VAR
	stValue: INT;
END_VAR
aRecipeParamsValues[0  ]:= DINT_TO_STRING(stActRecipe.stUBL.nRecipeIndexShow.diValue																		);
aRecipeParamsValues[1  ]:= DINT_TO_STRING(stActRecipe.stUBL.iPackageCapTypeShow.diValue																	);
aRecipeParamsValues[2  ]:= DINT_TO_STRING(stActRecipe.stUBL.iPackageCapDiameterShow.diValue 																);
aRecipeParamsValues[3  ]:= BOOL_TO_STRING(stActRecipe.stUBL.bExEnableShow.bValue 																			);
aRecipeParamsValues[4  ]:= BOOL_TO_STRING(stActRecipe.stUBL.bBottleFeederEnableShow.bValue																);
aRecipeParamsValues[5  ]:= UDINT_TO_STRING(stActRecipe.stUBL.iBottleFeederTurntableVelocitySVShow.udiValue														);
aRecipeParamsValues[6  ]:= DINT_TO_STRING(stActRecipe.stUBL.iBottleFeederBottleSensorDelayShow.diValue													);
aRecipeParamsValues[7  ]:= DINT_TO_STRING(stActRecipe.stUBL.iBottleFeederFormGateDelayShow.diValue														);
aRecipeParamsValues[8  ]:= DINT_TO_STRING(stActRecipe.stUBL.iBottleFeederAllowFormDelayShow.diValue														);
aRecipeParamsValues[9  ]:= BOOL_TO_STRING(stActRecipe.stUBL.bPucksInserterEnableShow.bValue																);
aRecipeParamsValues[10 ]:= UDINT_TO_STRING(stActRecipe.stUBL.iPucksInserterTurntableVelocitySVShow.udiValue 													);
aRecipeParamsValues[11 ]:= UDINT_TO_STRING(stActRecipe.stUBL.iPucksInserterConveyorVelocitySVShow.udiValue														);
aRecipeParamsValues[12 ]:= DINT_TO_STRING(stActRecipe.stUBL.iPucksInserterBottleSensorDelayShow.diValue													);
aRecipeParamsValues[13 ]:= DINT_TO_STRING(stActRecipe.stUBL.iPucksInserterFormGateDelayShow.diValue 														);
aRecipeParamsValues[14 ]:= DINT_TO_STRING(stActRecipe.stUBL.iPucksInserterAllowFormDelayShow.diValue 														);
aRecipeParamsValues[15 ]:= LREAL_TO_STRING(stActRecipe.stUBL.lrPucksInserterWheelOffsetShow.lrValue 															);
aRecipeParamsValues[16 ]:= LREAL_TO_STRING(stActRecipe.stUBL.lrPucksInserterWheelAccelerationShow.lrValue 														);
aRecipeParamsValues[17 ]:= LREAL_TO_STRING(stActRecipe.stUBL.lrPucksInserterWheelVelocityShow.lrValue 															);
aRecipeParamsValues[18 ]:= LREAL_TO_STRING(stActRecipe.stUBL.lrPucksInserterHammerHeightSVShow.lrValue 														);
aRecipeParamsValues[19 ]:= BOOL_TO_STRING(stActRecipe.stUBL.bGateBeforeDispencersEnableShow.bValue														);
aRecipeParamsValues[20 ]:= LREAL_TO_STRING(stActRecipe.stUBL.nGateBeforeDispencersTimeFormInsertingShow.lrValue 												);
aRecipeParamsValues[21 ]:= BOOL_TO_STRING(stActRecipe.stUBL.bGateAfterWeightEnableShow.bValue 															);
aRecipeParamsValues[22 ]:= LREAL_TO_STRING(stActRecipe.stUBL.nGateAfterWeightTimeFormInsertingShow.lrValue 													);
aRecipeParamsValues[25 ]:= BOOL_TO_STRING(stActRecipe.stUBL.bGateRobotEnableShow.bValue       															);
aRecipeParamsValues[26 ]:= LREAL_TO_STRING(stActRecipe.stUBL.nGateRobotTimeFormInsertingShow.lrValue															);
aRecipeParamsValues[27 ]:= BOOL_TO_STRING(stActRecipe.stUBL.bFormsDragingLeftEnableShow.bValue         													);
aRecipeParamsValues[28 ]:= LREAL_TO_STRING(stActRecipe.stUBL.lrFormsDragingLeftVelocityShow.lrValue         													);
aRecipeParamsValues[29 ]:= LREAL_TO_STRING(stActRecipe.stUBL.lrFormsDragingLeftAccelerationShow.lrValue 														);
aRecipeParamsValues[30 ]:= LREAL_TO_STRING(stActRecipe.stUBL.lrFormsDragingLeftDecelerationShow.lrValue   														);
aRecipeParamsValues[31 ]:= BOOL_TO_STRING(stActRecipe.stUBL.bFormsDragingRightEnableShow.bValue 															);
aRecipeParamsValues[32 ]:= LREAL_TO_STRING(stActRecipe.stUBL.lrFormsDragingRightVelocityShow.lrValue 															);
aRecipeParamsValues[33 ]:= LREAL_TO_STRING(stActRecipe.stUBL.lrFormsDragingRightAccelerationShow.lrValue 														);
aRecipeParamsValues[34 ]:= LREAL_TO_STRING(stActRecipe.stUBL.lrFormsDragingRightDecelerationShow.lrValue 														);
aRecipeParamsValues[35 ]:= BOOL_TO_STRING(stActRecipe.stUBL.bDosingTwoPhasesShow.bValue 	        														);
aRecipeParamsValues[36 ]:= LREAL_TO_STRING(stActRecipe.stUBL.lrDispencersLifterReadyPositionShow.lrValue 														);
aRecipeParamsValues[37 ]:= UDINT_TO_STRING(stActRecipe.stUBL.uiDispencerStartDosingDelayShow.udiValue 															);
aRecipeParamsValues[38 ]:= BOOL_TO_STRING(stActRecipe.stUBL.bDispencer1EnableShow.bValue 	          														);
aRecipeParamsValues[39 ]:= BOOL_TO_STRING(stActRecipe.stUBL.bDispencer2EnableShow.bValue 		  															);
aRecipeParamsValues[40 ]:= BOOL_TO_STRING(stActRecipe.stUBL.bDispencer3EnableShow.bValue           														);
aRecipeParamsValues[41 ]:= BOOL_TO_STRING(stActRecipe.stUBL.bDispencer4EnableShow.bValue 			       													);
aRecipeParamsValues[42 ]:= LREAL_TO_STRING(stActRecipe.stUBL.lrDispencer1DoseVolumeShow.lrValue 				   												);
aRecipeParamsValues[43 ]:= LREAL_TO_STRING(stActRecipe.stUBL.lrDispencer1Phase1VolumeShow.lrValue	           													);
aRecipeParamsValues[44 ]:= LREAL_TO_STRING(stActRecipe.stUBL.lrDispencer1Phase2VolumeShow.lrValue 	       														);
aRecipeParamsValues[45 ]:= LREAL_TO_STRING(stActRecipe.stUBL.lrDispencer1Phase1VelocityShow.lrValue 	       													);
aRecipeParamsValues[46 ]:= LREAL_TO_STRING(stActRecipe.stUBL.lrDispencer1Phase2VelocityShow.lrValue 															);
aRecipeParamsValues[47 ]:= LREAL_TO_STRING(stActRecipe.stUBL.lrDispencer1Phase3VelocityShow.lrValue 		   													);
aRecipeParamsValues[48 ]:= LREAL_TO_STRING(stActRecipe.stUBL.lrDispencer1SuckVelocityShow.lrValue   															);
aRecipeParamsValues[49 ]:= LREAL_TO_STRING(stActRecipe.stUBL.lrDispencer1Phase1AccelerationShow.lrValue 														);
aRecipeParamsValues[50 ]:= LREAL_TO_STRING(stActRecipe.stUBL.lrDispencer1Phase2AccelerationShow.lrValue 	  													);
aRecipeParamsValues[51 ]:= LREAL_TO_STRING(stActRecipe.stUBL.lrDispencer1Phase3AccelerationShow.lrValue 	   													);
aRecipeParamsValues[52 ]:= LREAL_TO_STRING(stActRecipe.stUBL.lrDispencer1SuckAccelerationShow.lrValue  														);
aRecipeParamsValues[53 ]:= LREAL_TO_STRING(stActRecipe.stUBL.lrDispencer1Phase1DecelerationShow.lrValue        												);
aRecipeParamsValues[54 ]:= LREAL_TO_STRING(stActRecipe.stUBL.lrDispencer1Phase2DecelerationShow.lrValue 														);
aRecipeParamsValues[55 ]:= LREAL_TO_STRING(stActRecipe.stUBL.lrDispencer1Phase3DecelerationShow.lrValue 	   													);
aRecipeParamsValues[56 ]:= UDINT_TO_STRING(stActRecipe.stUBL.udiDispencer1DosingDoneDelayTimeShow.udiValue 													);
aRecipeParamsValues[57 ]:= LREAL_TO_STRING(stActRecipe.stUBL.lrDispencer1SuckValveOpenVolumeShow.lrValue 														);
aRecipeParamsValues[58 ]:= LREAL_TO_STRING(stActRecipe.stUBL.lrDispencer1SuckValveOpenTimeDelayShow.lrValue 													);
aRecipeParamsValues[59 ]:= LREAL_TO_STRING(stActRecipe.stUBL.lrDispencer1SuckValveCloseVolumeShow.lrValue 														);
aRecipeParamsValues[60 ]:= LREAL_TO_STRING(stActRecipe.stUBL.lrDispencer1SuckValveCloseTimeDelayShow.lrValue 													);
aRecipeParamsValues[61 ]:= LREAL_TO_STRING(stActRecipe.stUBL.lrDispencer1DoseValveOpenVolumeShow.lrValue    													);
aRecipeParamsValues[62 ]:= LREAL_TO_STRING(stActRecipe.stUBL.lrDispencer1DoseValveOpenTimeAccShow.lrValue   													);           						
aRecipeParamsValues[63 ]:= LREAL_TO_STRING(stActRecipe.stUBL.lrDispencer1DoseValveCloseVolumeShow.lrValue    													);           						
aRecipeParamsValues[64 ]:= LREAL_TO_STRING(stActRecipe.stUBL.lrDispencer1DoseValveCloseTimeDecShow.lrValue 													);
aRecipeParamsValues[65 ]:= LREAL_TO_STRING(stActRecipe.stUBL.lrDispencer1DoseSuckingVolumeShow.lrValue 														);
aRecipeParamsValues[66 ]:= LREAL_TO_STRING(stActRecipe.stUBL.lrDispencer1DoseSuckingTimeDelayShow.lrValue 														);
aRecipeParamsValues[67 ]:= BOOL_TO_STRING(stActRecipe.stUBL.bDispencer1DoseSuckingShow.bValue 			       											);
aRecipeParamsValues[68 ]:= BOOL_TO_STRING(stActRecipe.stUBL.bDispencer1LiftSynchroPh1Show.bValue 															);
aRecipeParamsValues[69 ]:= BOOL_TO_STRING(stActRecipe.stUBL.bDispencer1LiftSynchroPh2Show.bValue 			   												);	      							
aRecipeParamsValues[70 ]:= BOOL_TO_STRING(stActRecipe.stUBL.bDispencer1LiftSynchroPh3Show.bValue 		       												);             					
aRecipeParamsValues[71 ]:= LREAL_TO_STRING(stActRecipe.stUBL.lrDispencer1LifterStartDosePositionShow.lrValue													);     						
aRecipeParamsValues[72 ]:= LREAL_TO_STRING(stActRecipe.stUBL.lrDispencer1LifterStopDosePositionShow.lrValue 													);       			
aRecipeParamsValues[73 ]:= LREAL_TO_STRING(stActRecipe.stUBL.lrDispencer1LifterVelocityShow.lrValue            												);	         			
aRecipeParamsValues[74 ]:= LREAL_TO_STRING(stActRecipe.stUBL.lrDispencer1LifterAccelerationShow.lrValue        												);        				
aRecipeParamsValues[75 ]:= LREAL_TO_STRING(stActRecipe.stUBL.lrDispencer1LifterDecelerationShow.lrValue 		    											);              				
aRecipeParamsValues[76 ]:= LREAL_TO_STRING(stActRecipe.stUBL.lrDispencer2DoseVolumeShow.lrValue	            												);              				
aRecipeParamsValues[77 ]:= LREAL_TO_STRING(stActRecipe.stUBL.lrDispencer2Phase1VolumeShow.lrValue 			    												);              				
aRecipeParamsValues[78 ]:= LREAL_TO_STRING(stActRecipe.stUBL.lrDispencer2Phase2VolumeShow.lrValue 			    												);               			
aRecipeParamsValues[79 ]:= LREAL_TO_STRING(stActRecipe.stUBL.lrDispencer2Phase1VelocityShow.lrValue 		    												);               			
aRecipeParamsValues[80 ]:= LREAL_TO_STRING(stActRecipe.stUBL.lrDispencer2Phase2VelocityShow.lrvalue 		    												);               			
aRecipeParamsValues[81 ]:= LREAL_TO_STRING(stActRecipe.stUBL.lrDispencer2Phase3VelocityShow.lrValue 		    												);	      		
aRecipeParamsValues[82 ]:= LREAL_TO_STRING(stActRecipe.stUBL.lrDispencer2SuckVelocityShow.lrValue     															);      				
aRecipeParamsValues[83 ]:= LREAL_TO_STRING(stActRecipe.stUBL.lrDispencer2Phase1AccelerationShow.lrValue 	        											);	         	
aRecipeParamsValues[84 ]:= LREAL_TO_STRING(stActRecipe.stUBL.lrDispencer2Phase2AccelerationShow.lrValue 	        											);         			
aRecipeParamsValues[85 ]:= LREAL_TO_STRING(stActRecipe.stUBL.lrDispencer2Phase3AccelerationShow.lrValue 		    											);	                                        			
aRecipeParamsValues[86 ]:= LREAL_TO_STRING(stActRecipe.stUBL.lrDispencer2SuckAccelerationShow.lrValue   														);                                          			
aRecipeParamsValues[87 ]:= LREAL_TO_STRING(stActRecipe.stUBL.lrDispencer2Phase1DecelerationShow.lrValue 														);                                          			
aRecipeParamsValues[88 ]:= LREAL_TO_STRING(stActRecipe.stUBL.lrDispencer2Phase2DecelerationShow.lrValue 														);            		              			
aRecipeParamsValues[89 ]:= LREAL_TO_STRING(stActRecipe.stUBL.lrDispencer2Phase3DecelerationShow.lrValue 														);           	                			
aRecipeParamsValues[90 ]:= UDINT_TO_STRING(stActRecipe.stUBL.udiDispencer2DosingDoneDelayTimeShow.udiValue 													);                                			
aRecipeParamsValues[91 ]:= LREAL_TO_STRING(stActRecipe.stUBL.lrDispencer2SuckValveOpenVolumeShow.lrValue 														);                               			
aRecipeParamsValues[92 ]:= LREAL_TO_STRING(stActRecipe.stUBL.lrDispencer2SuckValveOpenTimeDelayShow.lrValue 													);                      			
aRecipeParamsValues[93 ]:= LREAL_TO_STRING(stActRecipe.stUBL.lrDispencer2SuckValveCloseVolumeShow.lrValue														);      					
aRecipeParamsValues[94 ]:= LREAL_TO_STRING(stActRecipe.stUBL.lrDispencer2SuckValveCloseTimeDelayShow.lrValue 													);          			
aRecipeParamsValues[95 ]:= LREAL_TO_STRING(stActRecipe.stUBL.lrDispencer2DoseValveOpenVolumeShow.lrValue 														);         			       	
aRecipeParamsValues[96 ]:= LREAL_TO_STRING(stActRecipe.stUBL.lrDispencer2DoseValveOpenTimeAccShow.lrValue 														);					                  	
aRecipeParamsValues[97 ]:= LREAL_TO_STRING(stActRecipe.stUBL.lrDispencer2DoseValveCloseVolumeShow.lrValue 														);					                       	
aRecipeParamsValues[98 ]:= LREAL_TO_STRING(stActRecipe.stUBL.lrDispencer2DoseValveCloseTimeDecShow.lrValue														);					                       	
aRecipeParamsValues[99 ]:= LREAL_TO_STRING(stActRecipe.stUBL.lrDispencer2DoseSuckingVolumeShow.lrValue	    													);					                       	
aRecipeParamsValues[100]:=	LREAL_TO_STRING(stActRecipe.stUBL.lrDispencer2DoseSuckingTimeDelayShow.lrValue														);					                       	
aRecipeParamsValues[101]:=	BOOL_TO_STRING(stActRecipe.stUBL.bDispencer2DoseSuckingShow.bValue 	            											);					                       	
aRecipeParamsValues[102]:=	BOOL_TO_STRING(stActRecipe.stUBL.bDispencer2LiftSynchroPh1Show.bValue 	        												);					
aRecipeParamsValues[103]:=	BOOL_TO_STRING(stActRecipe.stUBL.bDispencer2LiftSynchroPh2Show.bValue 	        												);							
aRecipeParamsValues[104]:=	BOOL_TO_STRING(stActRecipe.stUBL.bDispencer2LiftSynchroPh3Show.bValue 	        												);					    
aRecipeParamsValues[105]:=	LREAL_TO_STRING(stActRecipe.stUBL.lrDispencer2LifterStartDosePositionShow.lrValue													);					    
aRecipeParamsValues[106]:=	LREAL_TO_STRING(stActRecipe.stUBL.lrDispencer2LifterStopDosePositionShow.lrValue 													);					
aRecipeParamsValues[107]:=	LREAL_TO_STRING(stActRecipe.stUBL.lrDispencer2LifterVelocityShow.lrValue        													);					
aRecipeParamsValues[108]:=	LREAL_TO_STRING(stActRecipe.stUBL.lrDispencer2LifterAccelerationShow.lrValue 														);					
aRecipeParamsValues[109]:=	LREAL_TO_STRING(stActRecipe.stUBL.lrDispencer2LifterDecelerationShow.lrValue 	    												);					
aRecipeParamsValues[110]:=	BOOL_TO_STRING(stActRecipe.stUBL.bDispencersCatchEnableShow.bValue             												);					
aRecipeParamsValues[111]:=	BOOL_TO_STRING(stActRecipe.stUBL.bDispencersCatchMaxPressureShow.bValue          												);					
aRecipeParamsValues[112]:=	LREAL_TO_STRING(stActRecipe.stUBL.lrDispencersCatchHeightSVShow.lrValue																);					
aRecipeParamsValues[113]:=	LREAL_TO_STRING(stActRecipe.stUBL.lrDispencersCatch1ClosedValueShow.lrValue          												);					
aRecipeParamsValues[114]:=	LREAL_TO_STRING(stActRecipe.stUBL.lrDispencersCatch1OpenValueShow.lrValue          													);					
aRecipeParamsValues[115]:=	LREAL_TO_STRING(stActRecipe.stUBL.lrDispencersCatch2ClosedValueShow.lrValue       													);						
aRecipeParamsValues[116]:=	LREAL_TO_STRING(stActRecipe.stUBL.lrDispencersCatch2OpenValueShow.lrValue	    													);					 
aRecipeParamsValues[117]:=	LREAL_TO_STRING(stActRecipe.stUBL.lrDispencersCatch3ClosedValueShow.lrValue         												);					
aRecipeParamsValues[118]:=	LREAL_TO_STRING(stActRecipe.stUBL.lrDispencersCatch3OpenValueShow.lrValue           												);					
aRecipeParamsValues[119]:=	LREAL_TO_STRING(stActRecipe.stUBL.lrDispencersCatch4ClosedValueShow.lrValue         												);					
aRecipeParamsValues[120]:=	LREAL_TO_STRING(stActRecipe.stUBL.lrDispencersCatch4OpenValueShow.lrValue															);					
aRecipeParamsValues[121]:=	LREAL_TO_STRING(stActRecipe.stUBL.lrDispencersCatchToleranceShow.lrValue 	        												);					
aRecipeParamsValues[122]:=	BOOL_TO_STRING(stActRecipe.stUBL.bTank1MixerEnableShow.bValue    																); 
aRecipeParamsValues[123]:=	BOOL_TO_STRING(stActRecipe.stUBL.bTankHeatingEnableShow.bValue   																);
aRecipeParamsValues[124]:= DINT_TO_STRING(stActRecipe.stUBL.iTankHeatingTempSVShow.diValue  																);
aRecipeParamsValues[125]:= BOOL_TO_STRING(stActRecipe.stUBL.bTank1PressureEnableShow.bValue																);
aRecipeParamsValues[126]:= BOOL_TO_STRING(stActRecipe.stUBL.bTank1SupplyPumpEnableShow.bValue                             								);
aRecipeParamsValues[127]:= BOOL_TO_STRING(stActRecipe.stUBL.bTank2SupplyPumpEnableShow.bValue                             								);
aRecipeParamsValues[128]:= UDINT_TO_STRING(stActRecipe.stUBL.uTank1LevelSetpointShow.udiValue                              									);
aRecipeParamsValues[129]:= UDINT_TO_STRING(stActRecipe.stUBL.uTank2LevelSetpointShow.udiValue                              									);
aRecipeParamsValues[130]:= BOOL_TO_STRING(stActRecipe.stUBL.bTank1LevelSignalInvertShow.bValue 	                        								);
aRecipeParamsValues[131]:= BOOL_TO_STRING(stActRecipe.stUBL.bTank2LevelSignalInvertShow.bValue 	                        								);
aRecipeParamsValues[132]:= BOOL_TO_STRING(stActRecipe.stUBL.bWeight1EnableShow.bValue                                     								);
aRecipeParamsValues[133]:= LREAL_TO_STRING(stActRecipe.stUBL.lrWeightMassSVShow.lrValue	                                									);
aRecipeParamsValues[134]:= DINT_TO_STRING(stActRecipe.stUBL.iWeight1ActuatorUpDelayShow.diValue 															);
aRecipeParamsValues[135]:= DINT_TO_STRING(stActRecipe.stUBL.iWeight2ActuatorUpDelayShow.diValue                           								);
aRecipeParamsValues[136]:= DINT_TO_STRING(stActRecipe.stUBL.iWeight3ActuatorUpDelayShow.diValue                           								);
aRecipeParamsValues[137]:= DINT_TO_STRING(stActRecipe.stUBL.iWeight4ActuatorUpDelayShow.diValue                           								);
aRecipeParamsValues[138]:= DINT_TO_STRING(stActRecipe.stUBL.iWeight5ActuatorUpDelayShow.diValue                           								);
aRecipeParamsValues[139]:= DINT_TO_STRING(stActRecipe.stUBL.iWeight6ActuatorUpDelayShow.diValue                           								);
aRecipeParamsValues[140]:= LREAL_TO_STRING(stActRecipe.stUBL.lrFormWeightShow.lrValue                                      									);
aRecipeParamsValues[141]:= LREAL_TO_STRING(stActRecipe.stUBL.lrMass1DensityShow.lrValue                                    									);
aRecipeParamsValues[142]:= LREAL_TO_STRING(stActRecipe.stUBL.lrMass2DensityShow.lrValue                                    									);
aRecipeParamsValues[143]:= LREAL_TO_STRING(stActRecipe.stUBL.lrCupWeightShow.lrValue                                       									);
aRecipeParamsValues[144]:= LREAL_TO_STRING(stActRecipe.stUBL.lrWholePackageWeightShow.lrValue 	                            									);
aRecipeParamsValues[145]:= LREAL_TO_STRING(stActRecipe.stUBL.lrWeight1MeasurmentCorrectionShow.lrValue	                    									);
aRecipeParamsValues[146]:= BOOL_TO_STRING(stActRecipe.stUBL.bDispencer1WeightCorrectionEnableShow.bValue                  								);
aRecipeParamsValues[147]:= BOOL_TO_STRING(stActRecipe.stUBL.bDispencer2WeightCorrectionEnableShow.bValue                  								);
aRecipeParamsValues[148]:= BOOL_TO_STRING(stActRecipe.stUBL.bDispencer3WeightCorrectionEnableShow.bValue                  								);
aRecipeParamsValues[149]:= BOOL_TO_STRING(stActRecipe.stUBL.bDispencer4WeightCorrectionEnableShow.bValue                  								);
aRecipeParamsValues[150]:= LREAL_TO_STRING(stActRecipe.stUBL.lrWeightUpperToleranceShow.lrValue                            									);
aRecipeParamsValues[151]:= LREAL_TO_STRING(stActRecipe.stUBL.lrWeightLowerToleranceShow.lrValue                            									);
aRecipeParamsValues[152]:= UDINT_TO_STRING(stActRecipe.stUBL.iWeightCorrectionNumberOfSamplesShow.udiValue                 									);
aRecipeParamsValues[153]:= BOOL_TO_STRING(stActRecipe.stUBL.bLidFeederEnableShow.bValue                 													);
aRecipeParamsValues[154]:= BOOL_TO_STRING(stActRecipe.stUBL.bLidFeederHeaterEnableShow.bValue                             								);
aRecipeParamsValues[155]:= LREAL_TO_STRING(stActRecipe.stUBL.lrLidFeederHeightPosSVShow.lrValue                            									);
aRecipeParamsValues[156]:= DINT_TO_STRING(stActRecipe.stUBL.iLidFeederHeatingTimeShow.diValue                             								);
aRecipeParamsValues[157]:= DINT_TO_STRING(stActRecipe.stUBL.iLidFeederTempHisteresisShow.diValue                          								);
aRecipeParamsValues[158]:= DINT_TO_STRING(stActRecipe.stUBL.iLidFeeder1TempSVShow.diValue 	                            								);
aRecipeParamsValues[159]:= DINT_TO_STRING(stActRecipe.stUBL.iLidFeeder2TempSVShow.diValue 	                            								);
aRecipeParamsValues[160]:= BOOL_TO_STRING(stActRecipe.stUBL.bLidFeederDragingStationEnableShow.bValue 	                								);
aRecipeParamsValues[161]:= LREAL_TO_STRING(stActRecipe.stUBL.lrLidFeederDragingStationVelocityShow.lrValue	                									);
aRecipeParamsValues[162]:= LREAL_TO_STRING(stActRecipe.stUBL.lrLidFeederDragingStationAccelerationShow.lrValue	            									);
aRecipeParamsValues[163]:= LREAL_TO_STRING(stActRecipe.stUBL.lrLidFeederDragingStationDecelerationShow.lrValue	            									);
aRecipeParamsValues[164]:= BOOL_TO_STRING(stActRecipe.stUBL.bLidPuttedCheckEnableShow.bValue                              								);
aRecipeParamsValues[165]:= LREAL_TO_STRING(stActRecipe.stUBL.lrLidPuttedCheckHeightSVShow.lrValue                          									);
aRecipeParamsValues[166]:= LREAL_TO_STRING(stActRecipe.stUBL.lrLidPuttedCheckPositionShow.lrValue                          									);
aRecipeParamsValues[167]:= LREAL_TO_STRING(stActRecipe.stUBL.lrLidPuttedCheckAreaShow.lrValue                              									);
aRecipeParamsValues[168]:= DINT_TO_STRING(stActRecipe.stUBL.iLidPuttedCheckProgramShow.diValue                            								);
aRecipeParamsValues[169]:= BOOL_TO_STRING(stActRecipe.stUBL.bLidSealerEnableShow.bValue                                   								);
aRecipeParamsValues[170]:= BOOL_TO_STRING(stActRecipe.stUBL.bLidSealerHeaterEnableShow.bValue 	                        								);
aRecipeParamsValues[171]:= DINT_TO_STRING(stActRecipe.stUBL.iLidSealerHeatingTimeShow.diValue	                            								);
aRecipeParamsValues[172]:= LREAL_TO_STRING(stActRecipe.stUBL.lrLidSealerPressureShow.lrValue                               									);
aRecipeParamsValues[173]:= LREAL_TO_STRING(stActRecipe.stUBL.lrLidSealerHeightPosSVShow.lrValue                            									);
aRecipeParamsValues[174]:= DINT_TO_STRING(stActRecipe.stUBL.iLidSealerTempHisteresisShow.diValue                          								);
aRecipeParamsValues[175]:= DINT_TO_STRING(stActRecipe.stUBL.iLidSealer1TempSVShow.diValue 	                            								);
aRecipeParamsValues[176]:= DINT_TO_STRING(stActRecipe.stUBL.iLidSealer2TempSVShow.diValue 	                            								);
aRecipeParamsValues[177]:= BOOL_TO_STRING(stActRecipe.stUBL.bLidSealerDragingStationEnableShow.bValue                     								);
aRecipeParamsValues[178]:= LREAL_TO_STRING(stActRecipe.stUBL.lrLidSealerDragingStationVelocityShow.lrValue 	            									);
aRecipeParamsValues[179]:= LREAL_TO_STRING(stActRecipe.stUBL.lrLidSealerDragingStationAccelerationShow.lrValue	            									);
aRecipeParamsValues[180]:= LREAL_TO_STRING(stActRecipe.stUBL.lrLidSealerDragingStationDecelerationShow.lrValue	            									);
aRecipeParamsValues[181]:= BOOL_TO_STRING(stActRecipe.stUBL.bCapFeederGateEnableShow.bValue 	                            								);
aRecipeParamsValues[182]:= DINT_TO_STRING(stActRecipe.stUBL.iCapFeederGateBlockingTimeShow.diValue 	                    								);
aRecipeParamsValues[183]:= BOOL_TO_STRING(stActRecipe.stUBL.bCapFeederEnableShow.bValue                                   								);
aRecipeParamsValues[184]:= LREAL_TO_STRING(stActRecipe.stUBL.lrCapFeederHeightPosSVShow.lrValue                            									);
aRecipeParamsValues[185]:= DINT_TO_STRING(stActRecipe.stUBL.iCapFeederTimeDelayOnShow.diValue                             								);
aRecipeParamsValues[186]:= DINT_TO_STRING(stActRecipe.stUBL.iCapFeederTimeDelayOffShow.diValue                            								);
aRecipeParamsValues[187]:= DINT_TO_STRING(stActRecipe.stUBL.iCapFeederTimeToEmptySleeveErrorShow.diValue                  								);
aRecipeParamsValues[188]:= BOOL_TO_STRING(stActRecipe.stUBL.bCapSorterOnlyWeightOKEnableShow.bValue                       								);
aRecipeParamsValues[189]:= BOOL_TO_STRING(stActRecipe.stUBL.bCapSorterDragEnableShow.bValue                               								);
aRecipeParamsValues[190]:= LREAL_TO_STRING(stActRecipe.stUBL.lrCapSorterDragVelocityShow.lrValue                           									);
aRecipeParamsValues[191]:= LREAL_TO_STRING(stActRecipe.stUBL.lrCapSorterDragAccelerationShow.lrValue 	                    									);
aRecipeParamsValues[192]:= LREAL_TO_STRING(stActRecipe.stUBL.lrCapSorterDragDecelerationShow.lrValue 	                    									);
aRecipeParamsValues[193]:= BOOL_TO_STRING(stActRecipe.stUBL.bCapPuttedCheckEnableShow.bValue                              								);
aRecipeParamsValues[194]:= LREAL_TO_STRING(stActRecipe.stUBL.lrCapPuttedCheckHeightPosSVShow.lrValue 	                    									);
aRecipeParamsValues[195]:= BOOL_TO_STRING(stActRecipe.stUBL.bGripperScrewer1EnableShow.bValue 	                        								);
aRecipeParamsValues[196]:= LREAL_TO_STRING(stActRecipe.stUBL.lrGripperScrewingTightTorqueShow.lrValue                      									);
aRecipeParamsValues[197]:= BOOL_TO_STRING(stActRecipe.stUBL.bGripperScrewer2EnableShow.bValue 	                        								);
aRecipeParamsValues[198]:= LREAL_TO_STRING(stActRecipe.stUBL.lrGripperScrewing2TightTorqueShow.lrValue	                    									);
aRecipeParamsValues[199]:= DINT_TO_STRING(stActRecipe.stUBL.iGripperScrewer1ToolShow.diValue                              								);
aRecipeParamsValues[200]:= LREAL_TO_STRING(stActRecipe.stUBL.lrGripperScrewer1VelocityShow.lrValue                         									);
aRecipeParamsValues[201]:= DINT_TO_STRING(stActRecipe.stUBL.nGripperScrewer1TightTimeShow.diValue	                        								);
aRecipeParamsValues[202]:= DINT_TO_STRING(stActRecipe.stUBL.iGripperScrewer1StartDelayShow.diValue	                    								);
aRecipeParamsValues[203]:= LREAL_TO_STRING(stActRecipe.stUBL.lrGripperScrewerReadyPositionShow.lrValue 	                									);
aRecipeParamsValues[204]:= LREAL_TO_STRING(stActRecipe.stUBL.lrGripperScrewerPushingCapPositionShow.lrValue 	            									);
aRecipeParamsValues[205]:= LREAL_TO_STRING(stActRecipe.stUBL.lrGripperScrewerScrewingCapPositionShow.lrValue               									);
aRecipeParamsValues[206]:= LREAL_TO_STRING(stActRecipe.stUBL.lrGripperScrewerPressureShow.lrValue                          									);
aRecipeParamsValues[207]:= LREAL_TO_STRING(stActRecipe.stUBL.lrGripperScrewerCatchPressureShow.lrValue 	                									);
aRecipeParamsValues[208]:= LREAL_TO_STRING(stActRecipe.stUBL.lrDispencerCatchPressureShow.lrValue                          									);
aRecipeParamsValues[209]:= LREAL_TO_STRING(stActRecipe.stUBL.lrGripperScrewerPressureExhaustLevelShow.lrValue              									);
aRecipeParamsValues[210]:= LREAL_TO_STRING(stActRecipe.stUBL.lrGripperScrewerCatchPressureExhaustLevelShow.lrValue         									);
aRecipeParamsValues[211]:= LREAL_TO_STRING(stActRecipe.stUBL.lrGripperScrewerTurnoversToFullScrewedShow.lrValue 	        									);
aRecipeParamsValues[212]:= LREAL_TO_STRING(stActRecipe.stUBL.lrGripperScrewerThreadPitchShow.lrValue                       									);
aRecipeParamsValues[213]:= LREAL_TO_STRING(stActRecipe.stUBL.lrGripperScrewerThreadTimesShow.lrValue                       									);
aRecipeParamsValues[214]:= DINT_TO_STRING(stActRecipe.stUBL.nGripperScrewerCatchHeightSVShow.diValue	                    								);
aRecipeParamsValues[215]:= BOOL_TO_STRING(stActRecipe.stUBL.bGripperScrewer1FindScrewShow.bValue                          								);
aRecipeParamsValues[216]:= BOOL_TO_STRING(stActRecipe.stUBL.bGripperScrewer1Option4Show.bValue                            								);
aRecipeParamsValues[217]:= LREAL_TO_STRING(stActRecipe.stUBL.lrGripperScrewer1FindingScrewDegreeShow.lrValue               									);
aRecipeParamsValues[218]:= BOOL_TO_STRING(stActRecipe.stUBL.bGripperScrewer1Option1Show.bValue	                        								);
aRecipeParamsValues[219]:= BOOL_TO_STRING(stActRecipe.stUBL.bGripperScrewer1Option2Show.bValue	                        								);
aRecipeParamsValues[220]:= BOOL_TO_STRING(stActRecipe.stUBL.bGripperScrewer1Option3Show.bValue	                        								);
aRecipeParamsValues[221]:= BOOL_TO_STRING(stActRecipe.stUBL.bGripperScrewer1Option5Show.bValue	                        								);
aRecipeParamsValues[222]:= BOOL_TO_STRING(stActRecipe.stUBL.bGripperScrewer1Option6Show.bValue	                        								);
aRecipeParamsValues[223]:= BOOL_TO_STRING(stActRecipe.stUBL.bGripperScrewer1Option7Show.bValue	                        								);
aRecipeParamsValues[224]:= BOOL_TO_STRING(stActRecipe.stUBL.bBottleDragingStationEnableShow.bValue 	                    								);
aRecipeParamsValues[225]:= LREAL_TO_STRING(stActRecipe.stUBL.lrBottleDragingStationVelocityShow.lrValue                    									);
aRecipeParamsValues[226]:= BOOL_TO_STRING(stActRecipe.stUBL.bCapCorrectCheckEnableShow.bValue 	                        								);
aRecipeParamsValues[227]:= LREAL_TO_STRING(stActRecipe.stUBL.lrCapCorrectCheckHeightPosSVShow.lrValue                      									);
aRecipeParamsValues[228]:= BOOL_TO_STRING(stActRecipe.stUBL.bCapCorrectCheckCameraEnableShow.bValue                       								);
aRecipeParamsValues[229]:= DINT_TO_STRING(stActRecipe.stUBL.iCapCorrectCheckCameraProgramShow.diValue 	                								);
aRecipeParamsValues[230]:= BOOL_TO_STRING(stActRecipe.stUBL.bBottleTransferEnableShow.bValue			                    								);
aRecipeParamsValues[231]:= UDINT_TO_STRING(stActRecipe.stUBL.nBottleTransferProgramShow.udiValue			                									);
aRecipeParamsValues[232]:= DINT_TO_STRING(stActRecipe.stUBL.iBottleTransferPickOffsetXShow.diValue                        								);
aRecipeParamsValues[233]:= DINT_TO_STRING(stActRecipe.stUBL.iBottleTransferPickOffsetYShow.diValue 	                    								);
aRecipeParamsValues[234]:= DINT_TO_STRING(stActRecipe.stUBL.iBottleTransferPickOffsetZShow.diValue                        								);
aRecipeParamsValues[235]:= DINT_TO_STRING(stActRecipe.stUBL.iBottleTransferPick2OffsetXShow.diValue                       								);
aRecipeParamsValues[236]:= DINT_TO_STRING(stActRecipe.stUBL.iBottleTransferPick2OffsetYShow.diValue 	                    								);
aRecipeParamsValues[237]:= DINT_TO_STRING(stActRecipe.stUBL.iBottleTransferPick2OffsetZShow.diValue                       								);
aRecipeParamsValues[238]:= DINT_TO_STRING(stActRecipe.stUBL.iBottleTransferPlace1OffsetXShow.diValue 	                    								);
aRecipeParamsValues[239]:= DINT_TO_STRING(stActRecipe.stUBL.iBottleTransferPlace1OffsetYShow.diValue 	                    								);
aRecipeParamsValues[240]:= DINT_TO_STRING(stActRecipe.stUBL.iBottleTransferPlace1OffsetZShow.diValue 	                    								);
aRecipeParamsValues[241]:= DINT_TO_STRING(stActRecipe.stUBL.iBottleTransferPlace2OffsetXShow.diValue 	                    								);
aRecipeParamsValues[242]:= DINT_TO_STRING(stActRecipe.stUBL.iBottleTransferPlace2OffsetYShow.diValue 	                    								);
aRecipeParamsValues[243]:= DINT_TO_STRING(stActRecipe.stUBL.iBottleTransferPlace2OffsetZShow.diValue 	                    								);
aRecipeParamsValues[244]:=	DINT_TO_STRING(stActRecipe.stUBL.iBottleTransferSpeedShow.diValue 	                            								);
aRecipeParamsValues[245]:= BOOL_TO_STRING(stActRecipe.stUBL.bBottleTransferInkJetEnableShow.bValue 	                    								);
aRecipeParamsValues[246]:= BOOL_TO_STRING(stActRecipe.stUBL.bBottleTransferPickOnlyOneShow.bValue                         								);
aRecipeParamsValues[247]:= BOOL_TO_STRING(stActRecipe.stUBL.bBottleTransferWeightEnableShow.bValue 	                    								);
aRecipeParamsValues[248]:= DINT_TO_STRING(stActRecipe.stUBL.iBottleTransferWeightIntervalShow.diValue	                    								);
aRecipeParamsValues[249]:= BOOL_TO_STRING(stActRecipe.stUBL.bBottleTransferRotateEnableShow.bValue 	                    								);
aRecipeParamsValues[250]:= BOOL_TO_STRING(stActRecipe.stUBL.bBadBottleConveyorEnableShow.bValue                           								);
aRecipeParamsValues[251]:= UDINT_TO_STRING(stActRecipe.stUBL.nBadBottleConveyorVelocitySVShow.udiValue 	                									);
aRecipeParamsValues[252]:= BOOL_TO_STRING(stActRecipe.stUBL.bLabelMachineEnableShow.bValue 	                            								);
aRecipeParamsValues[253]:= BOOL_TO_STRING(stActRecipe.stUBL.bExitTurnTable1EnableShow.bValue                              								);
aRecipeParamsValues[254]:= BOOL_TO_STRING(stActRecipe.stUBL.bExitConveyorEnableShow.bValue                                								);
aRecipeParamsValues[255]:= UDINT_TO_STRING(stActRecipe.stUBL.nExitConveyorVelocitySVShow.udiValue 	                        									);
aRecipeParamsValues[256]:= BOOL_TO_STRING(stActRecipe.stUBL.bFormTransportersEnableShow.bValue						    								);
aRecipeParamsValues[257]:= UDINT_TO_STRING(stActRecipe.stUBL.nFormTransportersDispencerVelocitySVShow.udiValue	            									);
aRecipeParamsValues[258]:= UDINT_TO_STRING(stActRecipe.stUBL.nFormTransportersScrewerVelocitySVShow.udiValue			    									);
aRecipeParamsValues[259]:= UDINT_TO_STRING(stActRecipe.stUBL.nFormTransportersBeforeScrewerVelocitySVShow.udiValue	        									);
aRecipeParamsValues[260]:= UDINT_TO_STRING(stActRecipe.stUBL.nFormTransportersSlowerVelocitySVShow.udiValue		 	    									);
aRecipeParamsValues[261]:= BOOL_TO_STRING(stActRecipe.stUBL.bCircularInkjetEnableShow.bValue	 	                        								);
aRecipeParamsValues[262]:= DINT_TO_STRING(stActRecipe.stUBL.iCircularInkjetSpeedShow.diValue	 	                        								);
aRecipeParamsValues[263]:= DINT_TO_STRING(stActRecipe.stUBL.iCircularInkjetDelayShow.diValue	 	                        								);
aRecipeParamsValues[264]:= DINT_TO_STRING(stActRecipe.stUBL.iCircularInkjetHoldShow.diValue	 	                        								);
aRecipeParamsValues[265]:= DINT_TO_STRING(stActRecipe.stUCF.iCapSorterProductType.diValue 	                            								);
aRecipeParamsValues[266]:= UDINT_TO_STRING(stActRecipe.stUCF.uiCapSorterIndexShow.udiValue 																	);
aRecipeParamsValues[267]:= BOOL_TO_STRING(stActRecipe.stUCF.bPresenceBottleEnableShow.bValue 	                            								);
aRecipeParamsValues[268]:= BOOL_TO_STRING(stActRecipe.stUCF.bCapSorterTransporterEnableShow.bValue														);
aRecipeParamsValues[269]:= DINT_TO_STRING(stActRecipe.stUCF.iCapSorterTransporterTankConveyorVelocityShow.diValue											);
aRecipeParamsValues[270]:= DINT_TO_STRING(stActRecipe.stUCF.iCapSorterTransporterStartDelayTimeShow.diValue												);
aRecipeParamsValues[271]:= UDINT_TO_STRING(stActRecipe.stUCF.udiCapSorterTransporterTimeProductOnSensorBeforeBrushShow.udiValue								);
aRecipeParamsValues[272]:= DINT_TO_STRING(stActRecipe.stUCF.iCapSorterTransporterEmptyingConveyorSpeedShow.diValue										);
aRecipeParamsValues[273]:= DINT_TO_STRING(stActRecipe.stUCF.iCapSorterTransporterVolumeOfCapsShow.diValue													);
aRecipeParamsValues[274]:= BOOL_TO_STRING(stActRecipe.stUCF.bCapSorterWheelEnableShow.bValue							    								);
aRecipeParamsValues[275]:= LREAL_TO_STRING(stActRecipe.stUCF.lrCapSorterWheelMoveAccelerationEmptyTableShow.lrValue	    									);
aRecipeParamsValues[276]:= LREAL_TO_STRING(stActRecipe.stUCF.lrCapSorterWheelMoveDecelerationEmptyTableShow.lrValue	    									);
aRecipeParamsValues[277]:= LREAL_TO_STRING(stActRecipe.stUCF.lrCapSorterWheelMoveSpeedEmptyTableShow.lrValue			    									);
aRecipeParamsValues[278]:= LREAL_TO_STRING(stActRecipe.stUCF.lrCapSorterWheelMoveAngleEmptyTableShow.lrValue			    									);
aRecipeParamsValues[279]:= LREAL_TO_STRING(stActRecipe.stUCF.lrCapSorterWheelJerkAngleEmptyTableShow.lrValue			    									);
aRecipeParamsValues[280]:= DINT_TO_STRING(stActRecipe.stUCF.iCapSorterWheelWaitingAfterRotationEmptyTableShow.diValue     								);
aRecipeParamsValues[281]:= LREAL_TO_STRING(stActRecipe.stUCF.lrCapSorterWheelMoveAccelerationFullTableShow.lrValue	        									);
aRecipeParamsValues[282]:= LREAL_TO_STRING(stActRecipe.stUCF.lrCapSorterWheelMoveDecelerationFullTableShow.lrValue	        									);
aRecipeParamsValues[283]:= LREAL_TO_STRING(stActRecipe.stUCF.lrCapSorterWheelMoveSpeedFullTableShow.lrValue			    									);
aRecipeParamsValues[284]:= LREAL_TO_STRING(stActRecipe.stUCF.lrCapSorterWheelMoveAngleFullyTableShow.lrValue			    									);
aRecipeParamsValues[285]:= LREAL_TO_STRING(stActRecipe.stUCF.lrCapSorterWheelJerkAngleFullTableShow.lrValue			    									);
aRecipeParamsValues[286]:= DINT_TO_STRING(stActRecipe.stUCF.iCapSorterWheelWaitingAfterRotationFullTableShow.diValue      								);
aRecipeParamsValues[287]:= LREAL_TO_STRING(stActRecipe.stUCF.lrCapSorterWheelMoveAccelerationHalfFullTableShow.lrValue     									);
aRecipeParamsValues[288]:= LREAL_TO_STRING(stActRecipe.stUCF.lrCapSorterWheelMoveDecelerationHalfFullTableShow.lrValue     									);
aRecipeParamsValues[289]:= LREAL_TO_STRING(stActRecipe.stUCF.lrCapSorterWheelMoveSpeedHalfFullTableShow.lrValue												);
aRecipeParamsValues[290]:= LREAL_TO_STRING(stActRecipe.stUCF.lrCapSorterWheelMoveAngleHalfFullyTableShow.lrValue												);
aRecipeParamsValues[291]:= LREAL_TO_STRING(stActRecipe.stUCF.lrCapSorterWheelJerkAngleHalfFullTableShow.lrValue												);
aRecipeParamsValues[292]:= DINT_TO_STRING(stActRecipe.stUCF.iCapSorterWheelWaitingAfterRotationHalfFullTableShow.diValue 									);
aRecipeParamsValues[293]:= BOOL_TO_STRING(stActRecipe.stUCF.bCapSorterCameraEnableShow.bValue                            									);
aRecipeParamsValues[294]:= BOOL_TO_STRING(stActRecipe.stUCF.bCapSorterRobotEnableShow.bValue                 			    								);
aRecipeParamsValues[295]:= LREAL_TO_STRING(stActRecipe.stUCF.lrCapSorterRobotPlace1PositionXShow.lrValue														);
aRecipeParamsValues[296]:= LREAL_TO_STRING(stActRecipe.stUCF.lrCapSorterRobotPlace1PositionYShow.lrValue														);
aRecipeParamsValues[297]:= LREAL_TO_STRING(stActRecipe.stUCF.lrCapSorterRobotPlace1PositionZShow.lrValue														);
aRecipeParamsValues[298]:= LREAL_TO_STRING(stActRecipe.stUCF.lrCapSorterRobotPlace1PositionCShow.lrValue														);
aRecipeParamsValues[299]:= DINT_TO_STRING(stActRecipe.stUCF.iCapSorterRobotPickElevationShow.diValue														);
aRecipeParamsValues[300]:= DINT_TO_STRING(stActRecipe.stUCF.iCapSorterRobotPickTimeShow.diValue															);
aRecipeParamsValues[301]:= DINT_TO_STRING(stActRecipe.stUCF.iCapSorterRobotVacuumActivationShow.diValue													);
aRecipeParamsValues[302]:= DINT_TO_STRING(stActRecipe.stUCF.iCapSorterRobotVacuumOffShow.diValue						    								);
aRecipeParamsValues[303]:= DINT_TO_STRING(stActRecipe.stUCF.iCapSorterRobotPlaceTimeShow.diValue															);
aRecipeParamsValues[304]:= DINT_TO_STRING(stActRecipe.stUCF.iCapSorterRobotTCP_PlaceOffsetShow.diValue			    									);
aRecipeParamsValues[305]:= DINT_TO_STRING(stActRecipe.stUCF.iCapSorterRobotAccelerationDecelerationShow.diValue	 										);
aRecipeParamsValues[306]:= DINT_TO_STRING(stActRecipe.stUCF.iCapSorterRobotGripperWatchdogShow.diValue			    									);
aRecipeParamsValues[307]:= DINT_TO_STRING(stActRecipe.stUCF.iCapSorterRobotParalaxCorrectionShow.diValue		    										);
aRecipeParamsValues[308]:= DINT_TO_STRING(stActRecipe.stUCF.iCapSorterRobotNumberToolShow.diValue		 													);
aRecipeParamsValues[309]:= DINT_TO_STRING(stActRecipe.stUCF.iCapSorterRobotPickPositionZShow.diValue 														);
aRecipeParamsValues[310]:= DINT_TO_STRING(stActRecipe.stUCF.iCapSorterRobotTCP_Lenght.diValue		 														);
aRecipeParamsValues[311]:= DINT_TO_STRING(stActRecipe.stUCF.iCapSorterRobotProductDiametr.diValue	 														);
aRecipeParamsValues[312]:= BOOL_TO_STRING(stActRecipe.stUCF.bCapSorterIntermediateTransporterEnableShow.bValue											);
aRecipeParamsValues[313]:= DINT_TO_STRING(stActRecipe.stUCF.iCapSorterIntermediateTransporterAutoSpeedShow.diValue										);
aRecipeParamsValues[314]:= DINT_TO_STRING(stActRecipe.stUCF.iCapSorterIntermediateTransporterManualSpeedShow.diValue										);
aRecipeParamsValues[315]:= DINT_TO_STRING(stActRecipe.stUCF.iCapSorterIntermediateTransporterEmptyingSpeedShow.diValue									);
aRecipeParamsValues[316]:= DINT_TO_STRING(stActRecipe.stUCF.iCapSorterIntermediateTransporterDelayCountTimeShow.diValue									);
aRecipeParamsValues[317]:= DINT_TO_STRING(stActRecipe.stUCF.iCapSorterIntermediateTransporterReverseTimeShow.diValue										);
aRecipeParamsValues[318]:= UDINT_TO_STRING(stActRecipe.stUCF.udiCapSorterIntermediateTransporterTimeProductOnSensorShow.udiValue 								);
aRecipeParamsValues[319]:= LREAL_TO_STRING(stActRecipe.stUCF.lrCapSorterIntermediateTransporterWheelAngleShow.lrValue											);
aRecipeParamsValues[320]:= BOOL_TO_STRING(stActRecipe.stUCF.bCapSorterIntermediateBrushEnableShow.bValue			 	    								);
aRecipeParamsValues[321]:= DINT_TO_STRING(stActRecipe.stUCF.iCapSorterIntermediateBrushAutoSpeedShow.diValue		 	    								);
aRecipeParamsValues[322]:= DINT_TO_STRING(stActRecipe.stUCF.iCapSorterIntermediateBrushManualSpeedShow.diValue		  									);
aRecipeParamsValues[323]:= DINT_TO_STRING(stActRecipe.stUCF.iCapSorterIntermediateBrushEmptyingSpeedShow.diValue	 	    								);
aRecipeParamsValues[324]:= LREAL_TO_STRING(stActRecipe.stUCF.lrCapSorterIntermediateBrushPositionHeightSVShow.lrValue 											);
aRecipeParamsValues[325]:= BOOL_TO_STRING(stActRecipe.stUCF.bCapSorterBrush1OnWheelEnableShow.bValue			  											);
aRecipeParamsValues[326]:= DINT_TO_STRING(stActRecipe.stUCF.iCapSorterBrush1OnWheelAutoSpeedShow.diValue		  											);
aRecipeParamsValues[327]:= DINT_TO_STRING(stActRecipe.stUCF.iCapSorterBrush1OnWheelManualSpeedShow.diValue		     									);
aRecipeParamsValues[328]:= DINT_TO_STRING(stActRecipe.stUCF.iCapSorterBrush1OnWheelEmptyingSpeedShow.diValue	  											);
aRecipeParamsValues[329]:= LREAL_TO_STRING(stActRecipe.stUCF.lrCapSorterBrush1OnWheelPositionHeightSVShow.lrValue   											);
aRecipeParamsValues[330]:= BOOL_TO_STRING(stActRecipe.stUCF.bCapSorterBrush2OnWheelEnableShow.bValue			 											);
aRecipeParamsValues[331]:= DINT_TO_STRING(stActRecipe.stUCF.iCapSorterBrush2OnWheelAutoSpeedShow.diValue		 											);
aRecipeParamsValues[332]:= DINT_TO_STRING(stActRecipe.stUCF.iCapSorterBrush2OnWheelManualSpeedShow.diValue	      										);
aRecipeParamsValues[333]:= DINT_TO_STRING(stActRecipe.stUCF.iCapSorterBrush2OnWheelEmptyingSpeedShow.diValue	   											);
aRecipeParamsValues[334]:= LREAL_TO_STRING(stActRecipe.stUCF.lrCapSorterBrush2OnWheelPositionHeightSVShow.lrValue   											);
aRecipeParamsValues[335]:= BOOL_TO_STRING(stActRecipe.stUCF.bCapSorterFeederEnableShow.bValue																);
aRecipeParamsValues[336]:= BOOL_TO_STRING(stActRecipe.stUCF.bCapSorterFeederEnableTubeError.bValue														);
aRecipeParamsValues[337]:= LREAL_TO_STRING(stActRecipe.stUCF.lrCapSorterFeederMover1InputPositionShow.lrValue													);
aRecipeParamsValues[338]:= LREAL_TO_STRING(stActRecipe.stUCF.lrCapSorterFeederMover2InputPositionShow.lrValue													);
aRecipeParamsValues[339]:= LREAL_TO_STRING(stActRecipe.stUCF.lrCapSorterFeederMover1OutputPositionShow.lrValue													);
aRecipeParamsValues[340]:= LREAL_TO_STRING(stActRecipe.stUCF.lrCapSorterFeederMover2OutputPositionShow.lrValue													);
aRecipeParamsValues[341]:= LREAL_TO_STRING(stActRecipe.stUCF.lrCapSorterFeederSlotDistanceShow.lrValue															);
aRecipeParamsValues[342]:= LREAL_TO_STRING(stActRecipe.stUCF.lrCapSorterFeederMoverSpeedShow.lrValue															);
aRecipeParamsValues[343]:= LREAL_TO_STRING(stActRecipe.stUCF.lrCapSorterFeederMoverAccelerationShow.lrValue    												);
aRecipeParamsValues[344]:= LREAL_TO_STRING(stActRecipe.stUCF.lrCapSorterFeederMoveJerkShow.lrValue																);
aRecipeParamsValues[345]:= BOOL_TO_STRING(stActRecipe.stUCF.bCapSorterPreScrewerEnableShow.bValue															);
aRecipeParamsValues[346]:= BOOL_TO_STRING(stActRecipe.stUCF.bCapSorterPreScrewerPicker1EnableShow.bValue           										);
aRecipeParamsValues[347]:= BOOL_TO_STRING(stActRecipe.stUCF.bCapSorterPreScrewerPicker2EnableShow.bValue           										);
aRecipeParamsValues[348]:= BOOL_TO_STRING(stActRecipe.stUCF.bCapSorterPreScrewerPicker3EnableShow.bValue          										);
aRecipeParamsValues[349]:= BOOL_TO_STRING(stActRecipe.stUCF.bCapSorterPreScrewerPicker4EnableShow.bValue          										);
aRecipeParamsValues[350]:= LREAL_TO_STRING(stActRecipe.stUCF.lrCapSorterPreScrewerPickZPositionShow.lrValue													);
aRecipeParamsValues[351]:= LREAL_TO_STRING(stActRecipe.stUCF.lrCapSorterPreScrewerCatcherReleseShow.lrValue													);
aRecipeParamsValues[352]:= LREAL_TO_STRING(stActRecipe.stUCF.lrCapSorterPreScrewerCapCatcherZPositionShow.lrValue												);
aRecipeParamsValues[353]:= LREAL_TO_STRING(stActRecipe.stUCF.lrCapSorterPreScrewerTopZPositionShow.lrValue														);
aRecipeParamsValues[354]:= LREAL_TO_STRING(stActRecipe.stUCF.lrCapSorterPreScrewerCartesianCatchZPositionShow.lrValue											);
aRecipeParamsValues[355]:= LREAL_TO_STRING(stActRecipe.stUCF.lrCapSorterPreScrewerStrawCatcherZPositionShow.lrValue											);
aRecipeParamsValues[356]:= LREAL_TO_STRING(stActRecipe.stUCF.LrCapSorterPreScrewerCheckStrawCatcherActuatorZPosition.lrValue 									);
aRecipeParamsValues[357]:= LREAL_TO_STRING(stActRecipe.stUCF.lrCapSorterPreScrewerScrewerStartZPositionShow.lrValue											);
aRecipeParamsValues[358]:= LREAL_TO_STRING(stActRecipe.stUCF.lrCapSorterPreScrewerGripperOpenPositionShow.lrValue												);
aRecipeParamsValues[359]:= LREAL_TO_STRING(stActRecipe.stUCF.lrCapSorterPreScrewerPlaceZPositionShow.lrValue													);
aRecipeParamsValues[360]:= LREAL_TO_STRING(stActRecipe.stUCF.lrCapSorterPreScrewerBendingDistanceShow.lrValue              									);
aRecipeParamsValues[361]:= LREAL_TO_STRING(stActRecipe.stUCF.lrCapSorterPreScrewerStrawInsertDistance.lrValue              									);
aRecipeParamsValues[362]:= LREAL_TO_STRING(stActRecipe.stUCF.lrCapSorterPreScrewerPickXMover1PositionShow.lrValue          									);
aRecipeParamsValues[363]:= LREAL_TO_STRING(stActRecipe.stUCF.lrCapSorterPreScrewerPickXMover2PositionShow.lrValue          									);
aRecipeParamsValues[364]:= LREAL_TO_STRING(stActRecipe.stUCF.lrCapSorterPreScrewerPlaceXPositionShow.lrValue		        									);
aRecipeParamsValues[365]:= LREAL_TO_STRING(stActRecipe.stUCF.lrCapSorterPreScrewerScrewFindingShow.lrValue	                									);
aRecipeParamsValues[366]:= LREAL_TO_STRING(stActRecipe.stUCF.lrCapSorterPreScrewerScrewDistanceShow.lrValue                									);
aRecipeParamsValues[367]:= LREAL_TO_STRING(stActRecipe.stUCF.lrCapSorterPreScrewerPickerSpeedShow.lrValue		            									);
aRecipeParamsValues[368]:= LREAL_TO_STRING(stActRecipe.stUCF.lrCapSorterPreScrewerPickerAccelerationShow.lrValue	        									);
aRecipeParamsValues[369]:= LREAL_TO_STRING(stActRecipe.stUCF.lrCapSorterPreScrewerPickerJerkShow.lrValue			        									);
aRecipeParamsValues[370]:= LREAL_TO_STRING(stActRecipe.stUCF.lrCapSorterPreScrewerCatcherSpeedShow.lrValue		            									);
aRecipeParamsValues[371]:= LREAL_TO_STRING(stActRecipe.stUCF.lrCapSorterPreScrewerCatcherAccelerationShow.lrValue          									);
aRecipeParamsValues[372]:= LREAL_TO_STRING(stActRecipe.stUCF.lrCapSorterPreScrewerCatcherJerkShow.lrValue		            									);
aRecipeParamsValues[373]:= LREAL_TO_STRING(stActRecipe.stUCF.lrCapSorterPreScrewerScrewSpeedShow.lrValue			        									);
aRecipeParamsValues[374]:= LREAL_TO_STRING(stActRecipe.stUCF.lrCapSorterPreScrewerScrewAccelerationShow.lrValue	        									);
aRecipeParamsValues[375]:= LREAL_TO_STRING(stActRecipe.stUCF.lrCapSorterPreScrewerScrewJerkShow.lrValue			        									);
aRecipeParamsValues[376]:= LREAL_TO_STRING(stActRecipe.stUCF.lrCapSorterPreScrewerCatcherCatchingPositionShow.lrValue      									);
aRecipeParamsValues[377]:= LREAL_TO_STRING(stActRecipe.stUCF.lrCapSorterPreScrewerCatcherPlacePositionShow.lrValue	        									);
aRecipeParamsValues[378]:= LREAL_TO_STRING(stActRecipe.stUCF.lrCapSorterPreScrewerCatcherHightSVShow.lrValue			    									);
aRecipeParamsValues[379]:= BOOL_TO_STRING(stActRecipe.stUCF.bCapSorterPreScrewerBottleCatcherEnableShow.bValue		    								);
aRecipeParamsValues[380]:= LREAL_TO_STRING(stActRecipe.stUCF.lrCapSorterPreScrewerBottleCatch1OpenValueShow.lrValue	    									);
aRecipeParamsValues[381]:= LREAL_TO_STRING(stActRecipe.stUCF.lrCapSorterPreScrewerBottleCatch1CloseValueShow.lrValue	    									);
aRecipeParamsValues[382]:= LREAL_TO_STRING(stActRecipe.stUCF.lrCapSorterPreScrewerBottleCatch2OpenValueShow.lrValue	    									);
aRecipeParamsValues[383]:= LREAL_TO_STRING(stActRecipe.stUCF.lrCapSorterPreScrewerBottleCatch2CloseValueShow.lrValue	    									);
aRecipeParamsValues[384]:= LREAL_TO_STRING(stActRecipe.stUCF.lrCapSorterPreScrewerBottleCatch3OpenValueShow.lrValue	    									);
aRecipeParamsValues[385]:= LREAL_TO_STRING(stActRecipe.stUCF.lrCapSorterPreScrewerBottleCatch3CloseValueShow.lrValue	    									);
aRecipeParamsValues[386]:= LREAL_TO_STRING(stActRecipe.stUCF.lrCapSorterPreScrewerBottleCatch4OpenValueShow.lrValue	                      					);
aRecipeParamsValues[387]:= LREAL_TO_STRING(stActRecipe.stUCF.lrCapSorterPreScrewerBottleCatch4CloseValueShow.lrValue	                      					);
aRecipeParamsValues[388]:= LREAL_TO_STRING(stActRecipe.stUCF.lrCapSorterPreScrewerBottleCatchToleranceValueShow.lrValue                      					);
aRecipeParamsValues[389]:= LREAL_TO_STRING(stActRecipe.stUCF.lrCapSorterPreScrewerCatchAngleOpenSV.lrValue                       								);
aRecipeParamsValues[390]:= LREAL_TO_STRING(stActRecipe.stUCF.lrCapSorterPreScrewerWaitInPlaceTimeShow.lrValue                                					);
aRecipeParamsValues[391]:= BOOL_TO_STRING(stActRecipe.stUCF.bCapSorterPreScrewerCatchAngleOpenEnaShow.bValue                                				);
aRecipeParamsValues[392]:= BOOL_TO_STRING(stActRecipe.stUCF.bCapSorterPreScrewerPoundedInCap.bValue                       								);
aRecipeParamsValues[393]:= LREAL_TO_STRING(stActRecipe.stUCF.lrCapSorterBottleHightShow.lrValue		                                      					);
aRecipeParamsValues[394]:= LREAL_TO_STRING(stActRecipe.stUCF.lrCapSorterBottleNeckHightShow.lrValue	                                      					);
aRecipeParamsValues[395]:= LREAL_TO_STRING(stActRecipe.stUCF.lrCapSorterCapHightShow.lrValue			                                      					);
aRecipeParamsValues[396]:= LREAL_TO_STRING(stActRecipe.stUCF.lrCapSorterCapNeckHightShow.lrValue		                                      					);
aRecipeParamsValues[397]:= LREAL_TO_STRING(stActRecipe.stUCF.lrCapSorterSpare1.lrValue                															);
aRecipeParamsValues[398]:= LREAL_TO_STRING(stActRecipe.stUCF.lrCapSorterSpare2.lrValue                															);
aRecipeParamsValues[399]:= LREAL_TO_STRING(stActRecipe.stUCF.lrCapSorterSpare3.lrValue                															);
aRecipeParamsValues[400]:= LREAL_TO_STRING(stActRecipe.stUCF.lrCapSorterSpare4.lrValue                															);
aRecipeParamsValues[401]:= LREAL_TO_STRING(stActRecipe.stUCF.lrCapSorterSpare5.lrValue                															);
aRecipeParamsValues[402]:= LREAL_TO_STRING(stActRecipe.stUCF.lrCapSorterSpare6.lrValue                															);
aRecipeParamsValues[403]:= LREAL_TO_STRING(stActRecipe.stUCF.lrCapSorterSpare7.lrValue                															);
aRecipeParamsValues[404]:= DINT_TO_STRING(stActRecipe.stUBF.iBottleSorterProductTypeShow.diValue                                            				);
aRecipeParamsValues[405]:= DINT_TO_STRING(stActRecipe.stUBF.uiBottleSorterIndexShow.diValue		                               							);
aRecipeParamsValues[406]:= BOOL_TO_STRING(stActRecipe.stUBF.bBottleSorterHopperTransporterEnableShow.bValue								  				);
aRecipeParamsValues[407]:= DINT_TO_STRING(stActRecipe.stUBF.iBottleSorterHopperConveyorRunningSpeedSVShow.diValue							  				);
aRecipeParamsValues[408]:= DINT_TO_STRING(stActRecipe.stUBF.iBottleSorterHopperConveyorEmptyingSpeedSVShow.diValue										);
aRecipeParamsValues[409]:= DINT_TO_STRING(stActRecipe.stUBF.iBottleSorterDistanceToFindElementOnTransferConveyorLimitRunningSVShow.diValue				);
aRecipeParamsValues[410]:= DINT_TO_STRING(stActRecipe.stUBF.iBottleSorterDistanceToFindElementOnTransferConveyorLimitEmptyingSVShow.diValue 				);
aRecipeParamsValues[411]:= BOOL_TO_STRING(stActRecipe.stUBF.bBottleSorterTransferTransporterEnableShow.bValue								  				);
aRecipeParamsValues[412]:= DINT_TO_STRING(stActRecipe.stUBF.iBottleSorterTransferConveyorRunningSpeedSVShow.diValue						  				);
aRecipeParamsValues[413]:= DINT_TO_STRING(stActRecipe.stUBF.iBottleSorterTransferConveyorEmptyingSpeedSVShow.diValue						  				);
aRecipeParamsValues[414]:= DINT_TO_STRING(stActRecipe.stUBF.iBottleSorterDistanceToFindElementOnSupplyConveyorDownstairsLimitSVShow.diValue 				);
aRecipeParamsValues[415]:= BOOL_TO_STRING(stActRecipe.stUBF.bBottleSorterSupplyTransporterEnableShow.bValue			                      				);
aRecipeParamsValues[416]:= UDINT_TO_STRING(stActRecipe.stUBF.uiBottleSorterSupplyTransporterRunningSpeedSVShow.udiValue                      					);
aRecipeParamsValues[417]:= UDINT_TO_STRING(stActRecipe.stUBF.uiBottleSorterSupplyTransporterEmptingSpeedSVShow.udiValue                      					);
aRecipeParamsValues[418]:= LREAL_TO_STRING(stActRecipe.stUBF.lrBottleSorterModuloMoveOffsetSVShow.lrValue				                      					);
aRecipeParamsValues[419]:= DINT_TO_STRING(stActRecipe.stUBF.iBottleSorterSensorsCountFirstConditionSVShow.diValue	                          				);
aRecipeParamsValues[420]:= DINT_TO_STRING(stActRecipe.stUBF.iBottleSorterSupplyTimeFirstConditionSVShow.diValue		                      				);
aRecipeParamsValues[421]:= DINT_TO_STRING(stActRecipe.stUBF.iBottleSorterSensorsCountSecondConditionMinSVShow.diValue	                      				);
aRecipeParamsValues[422]:= DINT_TO_STRING(stActRecipe.stUBF.iBottleSorterSensorsCountSecondConditionMaxSVShow.diValue	                      				);
aRecipeParamsValues[423]:= DINT_TO_STRING(stActRecipe.stUBF.iBottleSorterSupplyTimeSecondConditionSVShow.diValue		                      				);
aRecipeParamsValues[424]:= DINT_TO_STRING(stActRecipe.stUBF.iBottleSorterSensorsCountThirdConditionSVShow.diValue	                          				);
aRecipeParamsValues[425]:= DINT_TO_STRING(stActRecipe.stUBF.iBottleSorterSupplyTimeThirdConditionSVShow.diValue		                      				);
aRecipeParamsValues[426]:= BOOL_TO_STRING(stActRecipe.stUBF.bBottleSorterWeelEnableShow.bValue			                       							);
aRecipeParamsValues[427]:= LREAL_TO_STRING(stActRecipe.stUBF.lrBottleSorterWheelSpeedSVShow.lrValue			                             					);
aRecipeParamsValues[428]:= LREAL_TO_STRING(stActRecipe.stUBF.lrBottleSorterWheelEmptyingSpeedSVShow.lrValue	                              					);
aRecipeParamsValues[429]:= BOOL_TO_STRING(stActRecipe.stUBF.bBottleSorterBrushEnableShow.bValue			   												);
aRecipeParamsValues[430]:= LREAL_TO_STRING(stActRecipe.stUBF.lrBottleSorterBrushHeightPositionSVShow.lrValue                                 					);
aRecipeParamsValues[431]:= DINT_TO_STRING(stActRecipe.stUBF.iBottleSorterBrushRunningSpeedSVShow.diValue	                                  				);
aRecipeParamsValues[432]:= DINT_TO_STRING(stActRecipe.stUBF.iBottleSorterBrushEmptyingSpeedSVShow.diValue	                                  				);
aRecipeParamsValues[433]:= BOOL_TO_STRING(stActRecipe.stUBF.bBottleSorterRobotEnableShow.bValue	                            							);
aRecipeParamsValues[434]:= UDINT_TO_STRING(stActRecipe.stUBF.nBottleSorterRobotRecipeId.udiValue		                                						);
aRecipeParamsValues[435]:= LREAL_TO_STRING(stActRecipe.stUBF.lrBottleSorterRemainingTimeToSuctionShow.lrValue                                					);
aRecipeParamsValues[436]:= LREAL_TO_STRING(stActRecipe.stUBF.lrBottleSorterSuckerSuctionTimeShow.lrValue		                              					);
aRecipeParamsValues[437]:= LREAL_TO_STRING(stActRecipe.stUBF.lrBottleSorterRemainingTimeToRejectShow.lrValue                                 					);
aRecipeParamsValues[438]:= LREAL_TO_STRING(stActRecipe.stUBF.lrBottleSorterEjectorPulseShow.lrValue                                        					);
aRecipeParamsValues[439]:= LREAL_TO_STRING(stActRecipe.stUBF.lrBottleSorterZPickAboveTheBottleSVShow.lrValue	                              					);
aRecipeParamsValues[440]:= LREAL_TO_STRING(stActRecipe.stUBF.lrBottleSorterZPickMoveSVShow.lrValue			                            						);
aRecipeParamsValues[441]:= LREAL_TO_STRING(stActRecipe.stUBF.lrBottleSorterSafetyHeightSVShow.lrValue		                              						);
aRecipeParamsValues[442]:= BOOL_TO_STRING(stActRecipe.stUBF.bBottleSorterRecieverEnableShow.bValue			                              				);
aRecipeParamsValues[443]:= BOOL_TO_STRING(stActRecipe.stUBF.bBottleSorterRecieverSlot1EnableShow.bValue		                              				);
aRecipeParamsValues[444]:= BOOL_TO_STRING(stActRecipe.stUBF.bBottleSorterRecieverSlot2EnableShow.bValue		                              				);
aRecipeParamsValues[443]:= BOOL_TO_STRING(stActRecipe.stUBF.bBottleSorterRecieverSlot3EnableShow.bValue		                							);
aRecipeParamsValues[444]:= LREAL_TO_STRING(stActRecipe.stUBF.lrBottleSorterRecieverHeightPositionSVShow.lrValue                            					);
aRecipeParamsValues[445]:= LREAL_TO_STRING(stActRecipe.stUCF.lrCapSorterPreScrewerPickerSpeedWhenScrewerShow.lrValue										);
aRecipeParamsValues[446]:= BOOL_TO_STRING (stActRecipe.stUBL.bROPPCappingEnableShow.bValue																		);
aRecipeParamsValues[447]:= BOOL_TO_STRING (stActRecipe.stUBL.bROPPDragEnableShow.bValue	 				    													);
aRecipeParamsValues[448]:= BOOL_TO_STRING (stActRecipe.stUBL.bROPPFeederEnableShow.bValue																	);
aRecipeParamsValues[449]:= BOOL_TO_STRING (stActRecipe.stUBL.bROPPSlowerEnableShow.bValue	 																		);
aRecipeParamsValues[450]:= DINT_TO_STRING (stActRecipe.stUBL.iROPPCapping1ToolShow.diValue 				    														);
aRecipeParamsValues[451]:= DINT_TO_STRING (stActRecipe.stUBL.iROPPCappingTime2Show.diValue  				    														);
aRecipeParamsValues[452]:= DINT_TO_STRING (stActRecipe.stUBL.iROPPCappingTimeShow.diValue  				    														);
aRecipeParamsValues[453]:= DINT_TO_STRING (stActRecipe.stUBL.iROPPFeederTimeDelayOffShow.diValue 																);
aRecipeParamsValues[454]:= DINT_TO_STRING (stActRecipe.stUBL.iROPPFeederTimeDelayOnShow.diValue  																	);
aRecipeParamsValues[455]:= DINT_TO_STRING (stActRecipe.stUBL.iROPPFeederTimeToEmptySleeveErrorShow.diValue															);
aRecipeParamsValues[456]:= LREAL_TO_STRING(stActRecipe.stUBL.lrROPPCappingHeightPosSVShow.lrValue																	);
aRecipeParamsValues[457]:= LREAL_TO_STRING(stActRecipe.stUBL.lrROPPCappingVelocitySVShow.lrValue	 														);
aRecipeParamsValues[458]:= LREAL_TO_STRING(stActRecipe.stUBL.lrROPPDragAccelerationShow.lrValue	 		    												);
aRecipeParamsValues[459]:= LREAL_TO_STRING(stActRecipe.stUBL.lrROPPDragDecelerationShow.lrValue	 		    												);
aRecipeParamsValues[460]:= LREAL_TO_STRING(stActRecipe.stUBL.lrROPPDragVelocityShow.lrValue	 			    												);
aRecipeParamsValues[461]:= LREAL_TO_STRING(stActRecipe.stUBL.lrROPPFeederHeightPosSVShow.lrValue	 		            													);
aRecipeParamsValues[462]:= UDINT_TO_STRING(stActRecipe.stUBL.nROPPSlowerVelocitySVShow.udiValue			    													);
END_METHOD

METHOD METH_SetFactoryDefaults : BOOL
VAR_IN_OUT
	stPrcRecipe					:	ST_Recipe;
END_VAR
udiCurrentIndex																						:=		0;
wsCurrentCaption1																					:=		"Factory defaults";
wsCurrentCaption2																					:=		"-";

